FUNCTION_BLOCK TMS_Mover EXTENDS FB_Mover IMPLEMENTS ITmsMover
VAR
	_activateTrack : ActivateTrackForMover(_axis);
	mcReadTrackPositions : Tc3_McCollisionAvoidance.MC_ReadTrackPositions;
	axesMoveTo2 		: MoveModuloMoverToPosition(_axis) := (Gap := 100.0);
	_stOptions : ST_MoveAbsoluteCAOptions;
	ipTcIoXtsMover			: I_TcIoXtsXpuMover;
	stTmsActPositions			: ST_PositionInfo;
END_VAR

SUPER^();
IF _identInGroup <> 0 THEN
	mcReadTrackPositions(
		Axis:= THIS^._axis, 
		Enable:= TRUE, 
		Valid=> , 
		Busy=> , 
		TrackPosition=> , 
		TrackId=> , 
		PartPosition=> , 
		PartId=> , 
		Error=> , 
		ErrorId=> );
END_IF
_activateTrack();
IF _activateTrack.Done THEN 
	_stOptions.PositionReferenceSystem :=  _activateTrack.NewTrackId;
	axesMoveTo2.Options := _stOptions;
END_IF

IF ipTcIoXtsMover <> 0 THEN
	stTmsActPositions:=ipTcIoXtsMover.GetPositionInfo();
END_IF

axesMoveTo2();

METHOD ActivateTrack : BOOL
VAR_INPUT
	newTrack : OTCID;
END_VAR
IF NOT _activateTrack.Busy THEN
	_activateTrack.Execute(Track := newTrack);
	ActivateTrack := TRUE;
END_IF
END_METHOD

PROPERTY ActiveTrack : OTCID
GET
ActiveTrack := stTmsActPositions.nTrackObjectid;
END_GET
END_PROPERTY

METHOD PUBLIC HasCommand : BOOL
VAR_INPUT
END_VAR
HasCommand := axesMoveTo2.Busy;
END_METHOD

METHOD isAtPosition : BOOL
VAR_INPUT
	position : MC_LREAL;
END_VAR

VAR
	moduloPos: DINT;
END_VAR
//Create modulo position 
//moduloPos := LREAL_TO_DINT(stTmsActPositions.fTrackPosition) MOD LREAL_TO_DINT(_trackLength);
IF position > 1 THEN
	IF stTmsActPositions.fTrackPosition < position + 1 AND stTmsActPositions.fTrackPosition > position - 1 THEN
		isAtPosition := TRUE;
	END_IF  
ELSE
	IF stTmsActPositions.fTrackPosition < position + 1 AND stTmsActPositions.fTrackPosition > 0.0  
		OR stTmsActPositions.fTrackPosition < _trackLength AND stTmsActPositions.fTrackPosition > _trackLength - 1 THEN
		isAtPosition := TRUE;
	END_IF
END_IF
END_METHOD

METHOD PUBLIC isPastPosition : BOOL
VAR_INPUT
	position : MC_LREAL;
END_VAR
IF position > 1 THEN
	IF stTmsActPositions.fTrackPosition > position THEN
		isPastPosition := TRUE;
	END_IF  
END_IF
END_METHOD

METHOD PUBLIC MoveTo : BOOL
VAR_INPUT
	Position : MC_LREAL;
	Velocity : MC_LREAL;
	BackwardMove : BOOL;
END_VAR
IF NOT THIS^.isAtPosition(position := Position) THEN
	IF NOT axesMoveTo2.Busy THEN
		THIS^.axesMoveTo2.MoveTo(Position := Position, Velocity := Velocity, Direction := Tc2_MC2.MC_Direction.MC_Positive_Direction, Turns := 0);
		MoveTo := TRUE;
		_targetPos := Position;
	END_IF
END_IF
END_METHOD

METHOD PUBLIC SetMoverInterface : BOOL
VAR_INPUT
	MoverInterface : I_TcIoXtsXpuMover;
END_VAR
ipTcIoXtsMover := MoverInterface;
END_METHOD

END_FUNCTION_BLOCK

(* stored: Version 1.1.0.1, ProductVersion 3.1.4024.12
   POU TMS_Mover: Id {6b131325-7dfb-4240-b139-8c4216101462}, SpecialFunc None
   Method ActivateTrack: Id {5f8dc4a4-b7cd-44e5-baab-59a89ea4550d}
   Property ActiveTrack: Id {57a3c436-4ed1-47e6-9026-bef04c939162}
   Get Get: Id {c72e2ae2-e105-4edf-83a4-44deb2f5b1cf}
   Method HasCommand: Id {5a17fcc3-6110-4d5b-bc24-ae196e62ddf3}
   Method isAtPosition: Id {1cb134b7-8afd-4d69-a68f-d63401be7671}
   Method isPastPosition: Id {99c090fe-960e-4a77-8c44-cc361d9f893e}
   Method MoveTo: Id {cb5563f4-b88f-463c-953d-1f3d7238a315}
   Method SetMoverInterface: Id {c6449f51-a9d5-4b22-b175-863ee923058b} *)
